FUNCTION_BLOCK fbWeberUS_AI_Conversion
VAR_INPUT
	iAnalogInput : INT;
	iMaxValue : INT;
	iTargetPercentage : INT;
	i1stLimitRange : INT;
	i2ndLimitRange : INT;
	tDelayTime : TIME;
	bUsActivated	 : BOOL;



END_VAR
VAR_OUTPUT
	iPercent : INT;
	b1stLimitRange : BOOL;
	b2ndLimitRange : BOOL;

END_VAR
VAR
	rPersent: REAL;
	bAnalogInEN: BOOL;
	bMaxValueEN: BOOL;
	b1stLmitRangeEN: BOOL;
	b2ndLimitRangeEN: BOOL;
	TNR: TON;
	TPR: TON;
	bTargetPEN: BOOL;
	b1stBelowRangeINT: BOOL;
	b2ndAboveRangeINT: BOOL;
	b2ndBelowRangeINT: BOOL;
	b1stAboveRangeINT: BOOL;
END_VAR
VAR // added by the converter: edge detectors and wires of the graphical bodies
    _w1 : ANY;
    _w2, _w3 : BOOL;
END_VAR

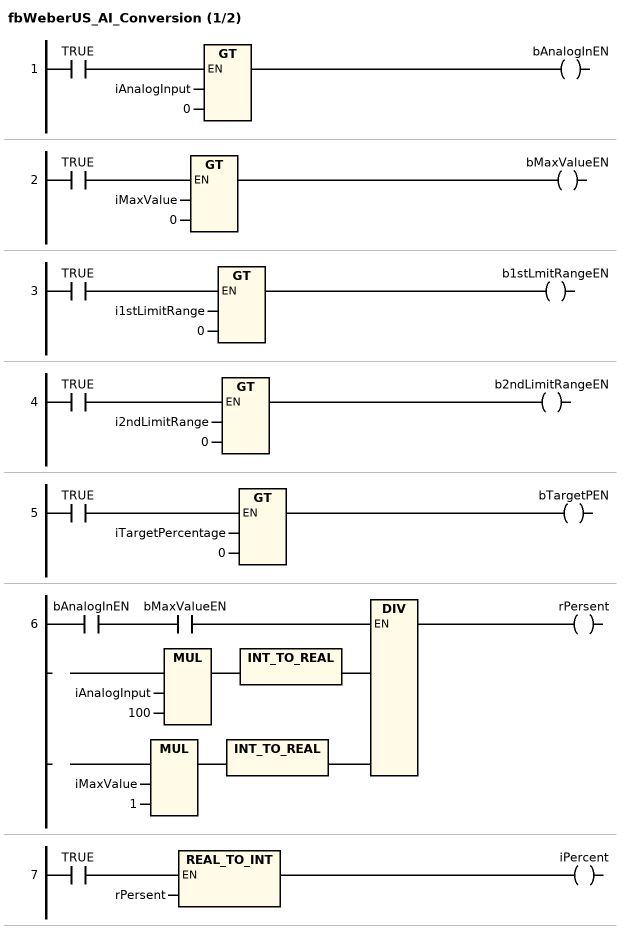
// NETWORK 1
bAnalogInEN := iAnalogInput > 0;

// NETWORK 2
bMaxValueEN := iMaxValue > 0;

// NETWORK 3
b1stLmitRangeEN := i1stLimitRange > 0;

// NETWORK 4
b2ndLimitRangeEN := i2ndLimitRange > 0;

// NETWORK 5
bTargetPEN := iTargetPercentage > 0;

// NETWORK 6
IF bAnalogInEN AND bMaxValueEN THEN _w1 := INT_TO_REAL(iAnalogInput * 100) / INT_TO_REAL(iMaxValue * 1); END_IF
rPersent := _w1;

// NETWORK 7
iPercent := REAL_TO_INT(rPersent);

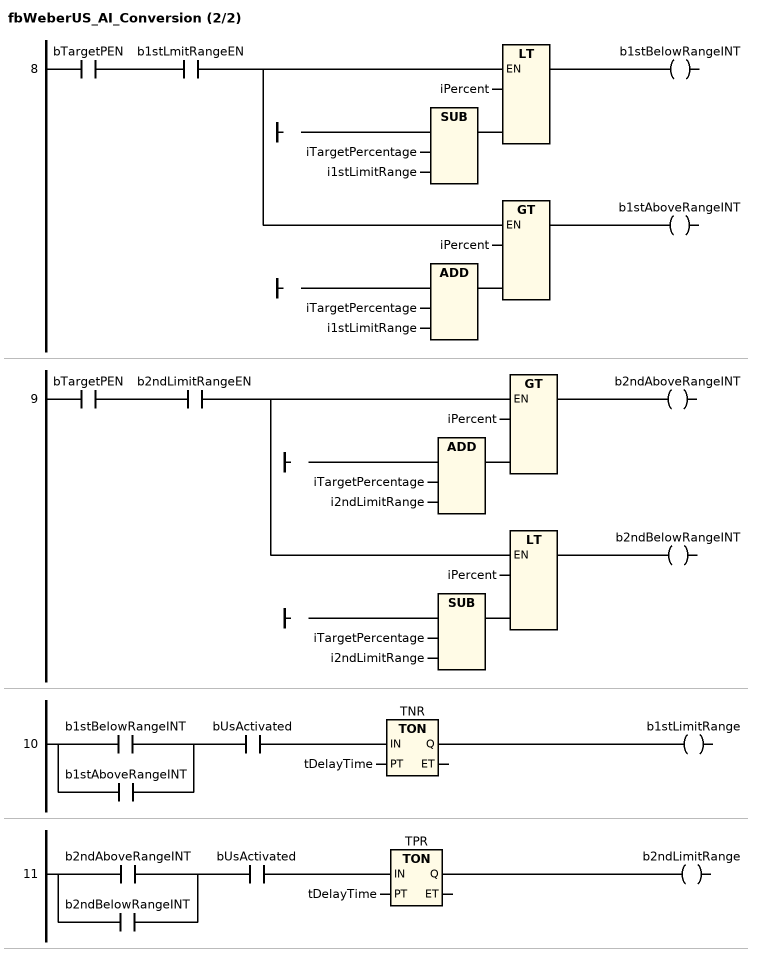
// NETWORK 8
_w2 := bTargetPEN AND b1stLmitRangeEN;
b1stBelowRangeINT := _w2 AND iPercent < iTargetPercentage - i1stLimitRange;
b1stAboveRangeINT := _w2 AND iPercent > iTargetPercentage + i1stLimitRange;

// NETWORK 9
_w3 := bTargetPEN AND b2ndLimitRangeEN;
b2ndAboveRangeINT := _w3 AND iPercent > iTargetPercentage + i2ndLimitRange;
b2ndBelowRangeINT := _w3 AND iPercent < iTargetPercentage - i2ndLimitRange;

// NETWORK 10
TNR(IN := (b1stBelowRangeINT OR b1stAboveRangeINT) AND bUsActivated, PT := tDelayTime); // TON
b1stLimitRange := TNR.Q;

// NETWORK 11
TPR(IN := (b2ndAboveRangeINT OR b2ndBelowRangeINT) AND bUsActivated, PT := tDelayTime); // TON
b2ndLimitRange := TPR.Q;

END_FUNCTION_BLOCK

(* stored: Version 1.1.0.1, ProductVersion 3.1.4024.12
   POU fbWeberUS_AI_Conversion: Id {e6ef03b6-2a27-4fc5-9129-34264e9a10da}, SpecialFunc None *)
